(* PLC project Unnamed, Unknown Unnamed 1 *)
(* stored: creationDateTime 2020-09-15T09:29:34, modificationDateTime 2023-06-14T00:00:00 *)

PROGRAM AutomaticDoorControl
  VAR
    Main_Switch AT %IX1.0 : BOOL;
    Object_Detection_Sensor AT %IX1.1 : BOOL;
    Open_Limit_Switch AT %IX1.2 : BOOL;
    Close_Limit_Switch AT %IX1.3 : BOOL;
    Open_Door_Motor AT %QX1.0 : BOOL;
    Close_Door_Motor AT %QX1.1 : BOOL;
    Door_Timer AT %TM1 : TON;
    Sequencer AT %IW1.0 : INT;
    Open_Switch_Count AT %IW2.0 : INT;
  END_VAR

            AutomaticDoorControl
            
              
                Main_Switch
              
              
                
                  
                    Sequencer
                    
                      0
                    
                  
                  
                    
                      
                        Close_Limit_Switch
                      
                      
                        
                          Open_Door_Motor
                          false
                        
                        
                          Close_Door_Motor
                          false
                        
                        
                          Sequencer
                          1
                        
                      
                    
                  
                
                
                  
                    Sequencer
                    
                      1
                    
                  
                  
                    
                      
                        
                          
                            Object_Detection_Sensor
                          
                          
                            
                              Open_Limit_Switch
                            
                          
                        
                      
                      
                        
                          Open_Door_Motor
                          true
                        
                        
                          Close_Door_Motor
                          false
                        
                      
                    
                    
                      
                        Open_Limit_Switch
                      
                      
                        
                          Open_Door_Motor
                          false
                        
                        
                          TON
                          Door_Timer
                          
                            
                              
                            
                            true
                          
                        
                        
                          Open_Switch_Count
                          Open_Switch_Count
                          +
                          1
                        
                        
                          
                            Open_Switch_Count
                            
                              5
                            
                            <
                          
                          
                            
                              Sequencer
                              2
                            
                          
                          
                            
                              
                                Sequencer
                                4
                              
                            
                          
                        
                      
                    
                  
                
                
                  
                    Sequencer
                    
                      2
                    
                  
                  
                    
                      
                        Door_Timer.Q
                      
                      
                        
                          Close_Door_Motor
                          true
                        
                        
                          TON
                          Door_Timer
                          
                            
                              
                            
                            false
                          
                        
                        
                          Sequencer
                          3
                        
                      
                    
                  
                
                
                  
                    Sequencer
                    
                      3
                    
                  
                  
                    
                      
                        Close_Limit_Switch
                      
                      
                        
                          Close_Door_Motor
                          false
                        
                        
                          Sequencer
                          1
                        
                      
                    
                  
                
                
                  
                    Sequencer
                    
                      4
                    
                  
                  
                    
                      
                        Open_Limit_Switch
                      
                      
                        
                          Open_Door_Motor
                          false
                        
                        
                          Close_Door_Motor
                          true
                        
                      
                      
                        
                          Close_Limit_Switch
                        
                        
                          
                            Close_Door_Motor
                            false
                          
                          
                            Open_Door_Motor
                            true
                          
                        
                      
                    
                  
                
              
            
          
END_PROGRAM

CONFIGURATION Config0
  RESOURCE Res0 ON PLC
    TASK task0(INTERVAL := T#20ms, PRIORITY := 0);
    PROGRAM instance0 WITH task0 : AutomaticDoorControl;
  END_RESOURCE
END_CONFIGURATION
